{attribute 'GeneratedUsingTerminal: EPP5151-0002-0016'}
{attribute addProperty BoxType "EPP5151-0002-0016"}
{attribute addProperty Description "EPP5151-0002 1Ch. Inc. Encoder 24V, M12, single ended"}
{attribute addProperty Physics "YY"}
{attribute addProperty Id "ENC_Status_compactAT %I*ENC_Status_compact_7D3464F320ENC_Control_compactAT %Q*ENC_Control_compact_21E2D14D6WcStateAT %I*WcState_9091E0EB2InfoDataAT %I*InfoData_32EB74EA10"}
{attribute addProperty CRC "1953950024"}
{attribute addProperty Size "38"}
TYPE EPP5151_7476E948 EXTENDS EtcSlaveBoxBase_77A0E4A7 :
STRUCT
	{attribute addProperty Name "ENC_Status_compact"}
	ENC_Status_compact : ENC_Status_compact_7D3464F3;
	{attribute addProperty Name "ENC_Control_compact"}
	ENC_Control_compact : ENC_Control_compact_21E2D14D;
	{attribute addProperty Name "WcState"}
	WcState : WcState_9091E0EB;
	{attribute addProperty Name "InfoData"}
	InfoData : InfoData_32EB74EA;
END_STRUCT
END_TYPE

(* stored: Version 1.2.0.0, ProductVersion 3.1.4024.11
   DUT EPP5151_7476E948: Id {566e09a2-d609-4592-b6fb-84f12263bda5} *)
